// TIA Portal V20 export
FUNCTION_BLOCK "LER_ServoPressHistory"   // FB201, LAD
// stored: Access Published, MemoryReserve 100, SetENOAutomatically false
   VAR_INPUT
      save : Bool;
      result : "LER_typePartData";
   END_VAR
   VAR_IN_OUT
      dataHistory : "LER_typeServoPressHistory";
   END_VAR
   VAR
      statDeleteData : "LER_typeServoPressHistory";
      statTrigger : Array[0..9] of Bool;
      statTonTimer : Array[0..99] of TON_TIME;
      statComplete : Bool;
   END_VAR
   VAR_TEMP
      tempRetVal : Array[0..9] of Int;
   END_VAR
   VAR_TEMP   // added for the SCL form of the ladder/FBD networks
      _w1 : Bool;
   END_VAR
BEGIN

REGION Network 1
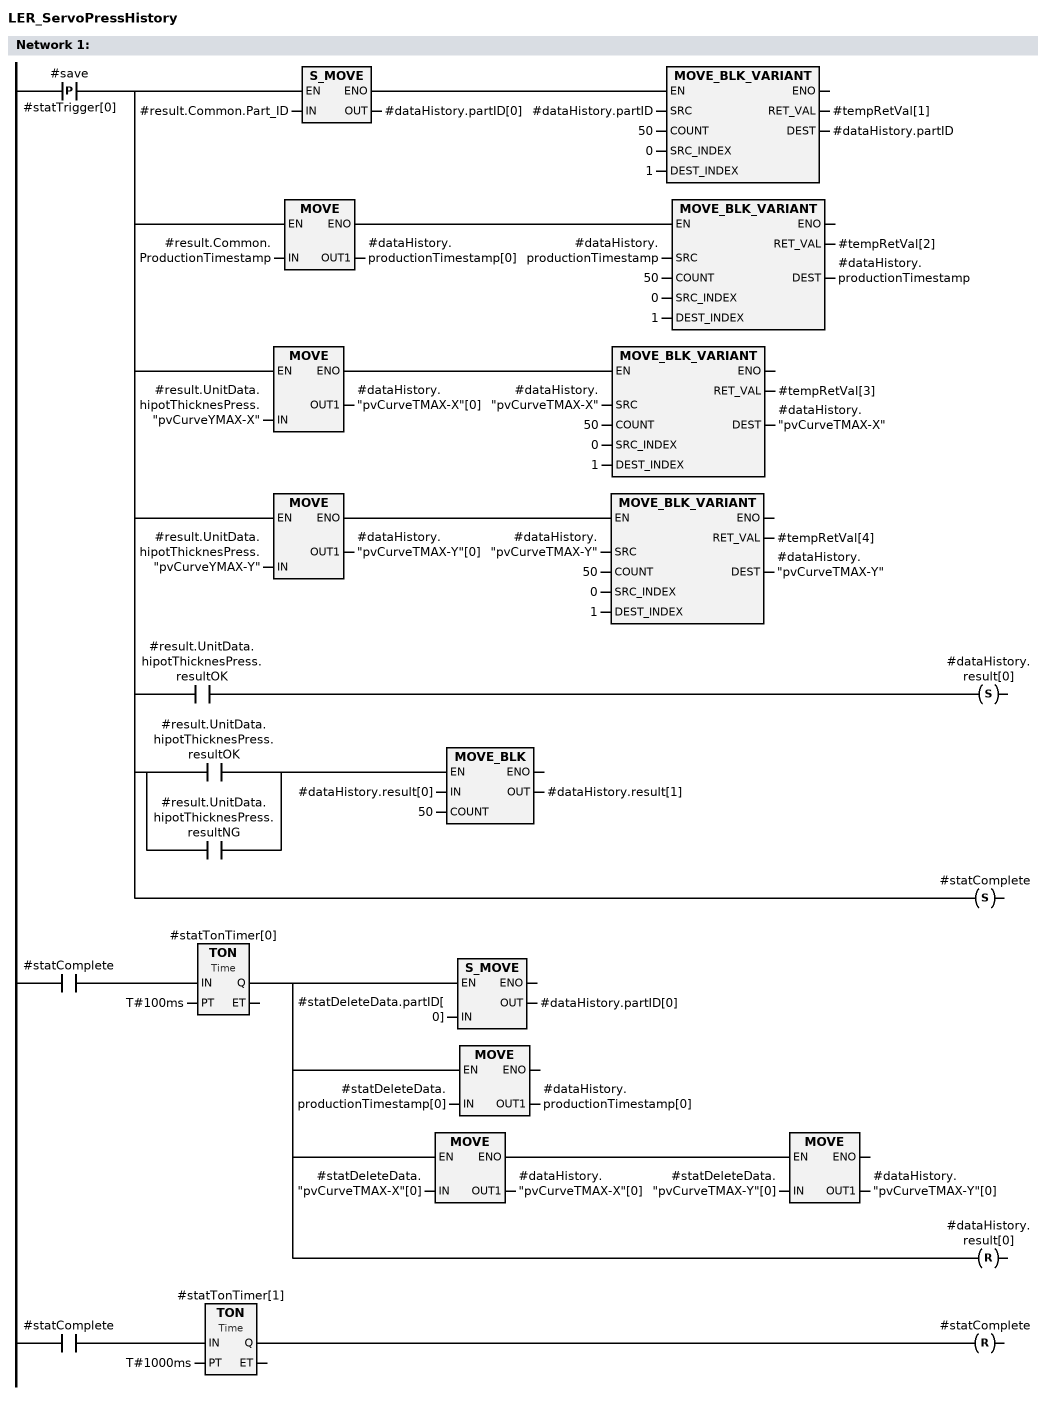
   #_w1 := #save AND NOT #statTrigger[0];   // rising edge of #save
   #statTrigger[0] := #save;
   IF #_w1 THEN
       #dataHistory.partID[0] := #result.Common.Part_ID;
       #tempRetVal[1] := MOVE_BLK_VARIANT(SRC := #dataHistory.partID,
                               COUNT := 50,
                               SRC_INDEX := 0,
                               DEST_INDEX := 1,
                               DEST => #dataHistory.partID);
       #dataHistory.productionTimestamp[0] := #result.Common.ProductionTimestamp;
       #tempRetVal[2] := MOVE_BLK_VARIANT(SRC := #dataHistory.productionTimestamp,
                               COUNT := 50,
                               SRC_INDEX := 0,
                               DEST_INDEX := 1,
                               DEST => #dataHistory.productionTimestamp);
       #dataHistory."pvCurveTMAX-X"[0] := #result.UnitData.hipotThicknesPress."pvCurveYMAX-X";
       #tempRetVal[3] := MOVE_BLK_VARIANT(SRC := #dataHistory."pvCurveTMAX-X",
                               COUNT := 50,
                               SRC_INDEX := 0,
                               DEST_INDEX := 1,
                               DEST => #dataHistory."pvCurveTMAX-X");
       #dataHistory."pvCurveTMAX-Y"[0] := #result.UnitData.hipotThicknesPress."pvCurveYMAX-Y";
       #tempRetVal[4] := MOVE_BLK_VARIANT(SRC := #dataHistory."pvCurveTMAX-Y",
                               COUNT := 50,
                               SRC_INDEX := 0,
                               DEST_INDEX := 1,
                               DEST => #dataHistory."pvCurveTMAX-Y");
   END_IF;
   IF #_w1 AND #result.UnitData.hipotThicknesPress.resultOK THEN #dataHistory.result[0] := TRUE; END_IF;
   IF #_w1 AND (#result.UnitData.hipotThicknesPress.resultOK OR #result.UnitData.hipotThicknesPress.resultNG) THEN
       MOVE_BLK(IN := #dataHistory.result[0], COUNT := 50, OUT => #dataHistory.result[1]);
   END_IF;
   IF #_w1 THEN #statComplete := TRUE; END_IF;
   #statTonTimer[0].TON(IN := #statComplete, PT := T#100ms);
   IF #statTonTimer[0].Q THEN
       #dataHistory.partID[0] := #statDeleteData.partID[0];
       #dataHistory.productionTimestamp[0] := #statDeleteData.productionTimestamp[0];
       #dataHistory."pvCurveTMAX-X"[0] := #statDeleteData."pvCurveTMAX-X"[0];
       #dataHistory."pvCurveTMAX-Y"[0] := #statDeleteData."pvCurveTMAX-Y"[0];
       #dataHistory.result[0] := FALSE;
   END_IF;
   #statTonTimer[1].TON(IN := #statComplete, PT := T#1000ms);
   IF #statTonTimer[1].Q THEN #statComplete := FALSE; END_IF;
END_REGION
END_FUNCTION_BLOCK
